// SIMATIC S7-200 project (STEP 7-Micro/WIN), CPU 226 REL 01.00

ORGANIZATION_BLOCK MAIN:OB1
TITLE= 项目注释：
// 
// 系统通过启动按钮1启动循环泵控制柜，控制循环泵1和循环泵2的运行，但循环泵1启动时，循环泵2不得同时运行，以避免电力过载。启动按钮3启动引风机控制柜，控制引风机；引风机启动前需确认循环泵运行标志置位，以确保炉内气流稳定。随后，鼓风机由启动按钮1触发，只有在引风机运行后才会启动，以维持炉内压力平衡。启动按钮2启动PLC控制柜，负责炉排电机、上煤电机、出渣电机和注油泵的运行。炉排电机由启动按钮2触发，需循环泵运行标志置位，以确保燃料供应；上煤电机只有在炉排电机运行后才会启动，以协调上煤和燃烧过程；出渣电机由启动按钮2控制，启动时不依赖炉排电机的状态。当上煤电机运行时，出渣电机可配合清除炉渣。注油泵在油压低时自动启动；延时定时器到时后，通过标志停止注油泵，以维持油压稳定。
// 系统通过多个传感器分别检测炉膛压力、炉膛温度、混合空气温度、排烟温度、进油温度和出油温度。当炉膛压力超过设定值时，触发报警标志；当炉膛温度高于设定值或低于设定值时，触发报警标志；炉膛温度低报警触发时，表示燃烧不足，上煤电机继续运行需谨慎。此时报警指示灯点亮；报警触发多个延时定时器，各定时器分别停止鼓风机、引风机、上煤电机和炉排电机，以安全停机。PID控制读取压力传感器和温度传感器的值，通过子程序调节炉膛压力和出油温度，确保工艺参数保持在设定范围内。操作员通过停止按钮1停止循环泵1，通过停止按钮2停止循环泵2；停止按钮3触发报警标志并点亮指示灯，保障操作安全。
// 
//  
BEGIN
Network 1 // 注油泵延时自动停止时间初始化
//  
// 
LD     SM0.1
MOVW   +1200, VW500
?000
Network 2 // 报警时间初始化
//  
// 
LD     SM0.1
MOVW   +300, VW502
Network 4 // 报警延时关断顺序初始化
// 
// 
LD     SM0.1
MOVW   +10, VW600
MOVW   +100, VW602
MOVW   +200, VW604
MOVW   +300, VW606
Network 5 // 报警延时关断顺序初始化
// 
// 
LDN    SM0.0
MOVW   +0, VW610
MOVW   +100, VW612
Network 7 // 炉膛报警压力设定
// 
// 
// 
LD     SM0.1
MOVW   -10000, VW1022
Network 8 // 炉膛报警温度高设定
// 
// 
LD     SM0.1
MOVW   +3000, VW1122
Network 9 // 炉膛报警温度低设定
// 
// 
// 
LD     SM0.1
MOVW   +1000, VW1124
Network 10 // 混合空气报警温度设定
// 
// 
LD     SM0.1
MOVW   +3000, VW1222
Network 11 // 排烟报警温度设定
// 
// 
LD     SM0.1
MOVW   +3000, VW1322
Network 12 // 出油报警温度高设定
// 
// 
// 
LD     SM0.1
MOVW   +3000, VW1522
Network 13 // 出油报警温度低设定
// 
// 
// 
LD     SM0.1
MOVW   +1000, VW1526
Network 15 // 模拟量设定值初始化--炉膛压力
// 
// 
LD     SM0.1
MOVW   -10000, VW1024
Network 16 // 模拟量设定值初始化--出油温度
// 
// 
LD     SM0.1
MOVW   +3000, VW1528
Network 18 // 循环泵控制柜－循环泵1
// 
// 
LD     I0.0
LPS
LD     M0.0
O      I0.3
O      T37
ALD
A      M0.2
AN     I0.5
AN     Q0.1
=      Q0.0
LPP
LPS
A      M0.0
S      M0.2, 1
LPP
A      M0.1
R      M0.2, 1
Network 19 // 泵1-延时等待运行信号
// 
// 
LD     Q0.0
EU
TOF    T37, +100
Network 20 // 循环泵控制柜－循环泵2
// 
// 
LD     I0.0
LPS
LD     M1.0
O      I0.4
O      T38
ALD
A      M1.2
AN     I0.6
AN     Q0.0
=      Q0.1
LPP
LPS
A      M1.0
S      M1.2, 1
LPP
A      M1.1
R      M1.2, 1
Network 21 // 泵2-延时等待运行信号
// 
// 
LD     Q0.1
EU
TOF    T38, +100
Network 22 // 循环泵启动信号
// 
// 
LD     Q0.0
O      Q0.1
=      M1.7
Network 24 // 引风机控制柜－引风机
// 
// 
LD     I0.2
LPS
LD     M2.0
O      I1.1
LDN    M2.1
O      Q0.5
ALD
ALD
AN     I1.2
A      M1.7
AN     T51
=      Q0.3
LPP
A      M2.2
=      Q0.2
Network 25 // 循环泵控制柜－鼓风机
//  
// 
//  
// 
LD     I0.0
LPS
LD     M3.0
O      I0.7
ALD
AN     M3.1
AN     I1.0
A      Q0.3
A      M1.7
AN     T50
=      Q0.5
LPP
A      M3.2
=      Q0.4
Network 27 // PLC控制柜－炉排电机
// 
// 
LD     I0.1
LD     M4.0
O      I2.0
ALD
LDN    M4.1
O      Q0.7
ALD
AN     I2.1
A      M1.7
AN     T53
=      Q0.6
Network 28 // PLC控制柜-上煤电机
// 
// 
LD     I0.1
LD     M5.0
O      I2.3
ALD
AN     M5.1
AN     I2.4
A      Q0.6
A      M1.7
AN     T52
=      Q0.7
Network 30 // PLC控制柜－出渣电机
// 
// 
LD     I0.1
LD     M6.0
O      I2.5
ALD
AN     M6.1
AN     I2.6
=      Q1.0
Network 31 // PLC控制柜－注油泵
// 
// 
LD     I0.1
LD     M7.0
O      I3.2
O      I3.1
ALD
AN     M7.1
AN     I3.3
AN     I3.0
AN     M7.7
=      Q1.1
Network 32
LD     I3.1
TOF    T39, VW500
Network 33
LD     T39
ED
=      M7.7
Network 35 // 模拟量读取/显示--炉膛压力
// 
// 
LDW<=  AIW4, +6500
MOVW   +6500, VW1000
Network 36
LDW>=  AIW4, +6500
AW<=   AIW4, +32000
MOVW   AIW4, VW1000
Network 37
LDW>=  AIW4, +32000
MOVW   +32000, VW1000
Network 38 // 炉膛压力线性运算
// 
// 
LD     SM0.0
MOVW   VW1000, VW1002
AENO
-I     +6500, VW1002
AENO
ITD    VW1002, VD1004
AENO
DTR    VD1004, VD1008
AENO
MOVR   VD1008, VD1012
AENO
/R     160.0, VD1012
AENO
ROUND  VD1012, VD1016
AENO
DTI    VD1016, VW1020
AENO
*I     -1, VW1020
Network 40 // 模拟量读取/显示--炉膛温度
// 
// 
LDW<=  AIW6, +6500
MOVW   +6500, VW1100
Network 41
LDW>=  AIW6, +6500
AW<=   AIW6, +32000
MOVW   AIW6, VW1100
Network 42
LDW>=  AIW6, +32000
MOVW   +32000, VW1100
Network 43 // 炉膛温度线性运算
// 
// 
// 
LD     SM0.0
MOVW   VW1100, VW1102
AENO
-I     +6500, VW1102
AENO
ITD    VW1102, VD1104
AENO
DTR    VD1104, VD1108
AENO
MOVR   VD1108, VD1112
AENO
/R     51.0, VD1112
AENO
ROUND  VD1112, VD1116
AENO
DTI    VD1116, VW1120
Network 45 // 模拟量读取/显示--混合空气温度
// 
// 
LDW<=  AIW8, +6500
MOVW   +6500, VW1200
Network 46
LDW>=  AIW8, +6500
AW<=   AIW8, +32000
MOVW   AIW8, VW1200
Network 47
LDW>=  AIW8, +32000
MOVW   +32000, VW1200
Network 48 // 炉膛温度线性运算
// 
// 
// 
LD     SM0.0
MOVW   VW1200, VW1202
AENO
-I     +6500, VW1202
AENO
ITD    VW1202, VD1204
AENO
DTR    VD1204, VD1208
AENO
MOVR   VD1208, VD1212
AENO
/R     51.0, VD1212
AENO
ROUND  VD1212, VD1216
AENO
DTI    VD1216, VW1220
Network 50 // 模拟量读取/显示--排烟温度
// 
// 
LDW<=  AIW10, +6500
MOVW   +6500, VW1300
Network 51
LDW>=  AIW10, +6500
AW<=   AIW10, +32000
MOVW   AIW10, VW1300
Network 52
LDW>=  AIW10, +32000
MOVW   +32000, VW1300
Network 53 // 排烟温度线性运算
// 
// 
// 
LD     SM0.0
MOVW   VW1300, VW1302
AENO
-I     +6500, VW1302
AENO
ITD    VW1302, VD1304
AENO
DTR    VD1304, VD1308
AENO
MOVR   VD1308, VD1312
AENO
/R     51.0, VD1312
AENO
ROUND  VD1312, VD1316
AENO
DTI    VD1316, VW1320
Network 55 // 模拟量读取/显示--进油温度
// 
// 
LDW<=  AIW12, +6500
MOVW   +6500, VW1400
Network 56
LDW>=  AIW12, +6500
AW<=   AIW12, +32000
MOVW   AIW12, VW1400
Network 57
LDW>=  AIW12, +32000
MOVW   +32000, VW1400
Network 58 // 进油温度线性运算
// 
// 
// 
LD     SM0.0
MOVW   VW1400, VW1402
AENO
-I     +6500, VW1402
AENO
ITD    VW1402, VD1404
AENO
DTR    VD1404, VD1408
AENO
MOVR   VD1408, VD1412
AENO
/R     51.0, VD1412
AENO
ROUND  VD1412, VD1416
AENO
DTI    VD1416, VW1420
Network 60 // 模拟量读取/显示--出油温度
// 
// 
LDW<=  AIW14, +6500
MOVW   +6500, VW1500
Network 61
LDW>=  AIW14, +6500
AW<=   AIW14, +32000
MOVW   AIW14, VW1500
Network 62
LDW>=  AIW14, +32000
MOVW   +32000, VW1500
Network 63 // 出油温度线性运算
// 
// 
// 
LD     SM0.0
MOVW   VW1500, VW1502
AENO
-I     +6500, VW1502
AENO
ITD    VW1502, VD1504
AENO
DTR    VD1504, VD1508
AENO
MOVR   VD1508, VD1512
AENO
/R     51.0, VD1512
AENO
ROUND  VD1512, VD1516
AENO
DTI    VD1516, VW1520
Network 65 // 炉膛负压报警控制
// 
// 
LDW>=  VW1020, VW1022
=      M8.0
Network 66
LDW<=  VW1022, -20000
=      M10.0
MOVW   -20000, VW1022
Network 67
LDW>=  VW1022, +0
=      M10.1
MOVW   +0, VW1022
Network 68 // 炉膛温度高报警控制
// 
// 
LDW>=  VW1120, VW1122
=      M8.1
Network 69
LDW>=  VW1122, +5000
=      M10.2
MOVW   +5000, VW1122
Network 70 // 炉膛温度低报警控制
// 
// 
LDW<=  VW1120, VW1124
=      M8.2
Network 71
LDW>=  VW1124, +5000
=      M10.3
MOVW   +5000, VW1224
Network 72
LDW>=  VW1124, VW1122
=      M10.4
MOVW   VW1122, VW1124
Network 73 // 混合空气温度报警控制
// 
// 
LDW>=  VW1220, VW1222
=      M8.3
Network 74
LDW>=  VW1222, +5000
=      M10.5
MOVW   +5000, VW1222
Network 75 // 排烟报警温度控制
// 
// 
LDW>=  VW1320, VW1322
=      M8.4
Network 76
LDW>=  VW1322, +5000
=      M10.6
MOVW   +5000, VW1322
Network 77 // 出油温度报警控制
// 
// 
LD     SM0.0
MOVW   VW1522, VW1524
+I     +6, VW1524
Network 78
// 
// 
LDW>=  VW1520, VW1524
=      M8.5
Network 79
LDW>=  VW1522, +5000
=      M10.7
MOVW   +5000, VW1522
Network 80
// 
// 
LDW<=  VW1520, VW1526
=      M8.6
Network 81
LDW>=  VW1526, +5000
=      M11.0
MOVW   +5000, VW1526
Network 82
LDW>=  VW1526, VW1522
=      M11.1
MOVW   VW1522, VW1526
Network 84 // 报警控制
// 
// 
LD     I0.5
EU
LD     I0.6
EU
OLD
LD     I1.0
EU
OLD
LD     I1.2
EU
OLD
LD     I1.5
EU
OLD
LD     I1.6
EU
OLD
LD     I2.1
EU
OLD
LD     I2.4
EU
OLD
LD     I2.6
EU
OLD
LD     I3.0
EU
OLD
LD     I3.1
EU
OLD
LD     I3.3
EU
OLD
LD     M8.0
EU
OLD
LD     M8.1
EU
OLD
LD     M8.2
EU
OLD
LD     M8.3
EU
OLD
LD     M8.4
EU
OLD
LD     M8.5
EU
OLD
LD     M8.6
EU
OLD
TOF    T40, VW502
S      M9.0, 1
Network 85 // 报警声音控制
// 
// 
LDN    T42
TON    T41, +10
Network 86
LD     T41
TON    T42, +10
Network 87 // 报警控制
// 
// 
LD     I0.5
O      I0.6
O      I1.0
O      I1.2
O      I1.5
O      I1.6
O      I2.1
O      I2.4
O      I2.6
O      I3.0
O      I3.1
O      I3.3
O      M8.0
O      M8.1
O      M8.2
O      M8.3
O      M8.4
O      M8.5
O      M8.6
A      M9.0
A      T40
AN     T42
=      Q1.2
Network 88 // 消音
// 
// 
LD     M9.1
R      M9.0, 1
Network 90 // 故障停机顺序
// 
// 
LD     M8.0
O      M8.1
O      M8.5
O      I1.5
O      I1.6
TON    T50, VW600
TON    T51, VW602
TON    T52, VW604
TON    T53, VW606
Network 91 // 进/出口油压高故障停机顺序控制
// 
// 
LDN    SM0.0
LD     I1.5
O      I1.6
ALD
TON    T55, VW610
TON    T56, VW612
Network 93 // PID模拟量设定值--炉膛压力设定
// 
// 
LD     SM0.0
ITD    VW1024, VD1026
AENO
DTR    VD1026, VD1030
AENO
MOVW   VW1030, VW104
/I     -20000, VW104
Network 94
LDW<=  VW1024, -20000
=      M11.2
MOVW   -20000, VW1024
Network 95
LDW>=  VW1024, +0
=      M11.3
MOVW   +0, VW1024
Network 96 // PID模拟量设定值--出油温度设定
// 
// 
LD     SM0.0
ITD    VW1528, VD1530
AENO
DTR    VD1530, VD1534
AENO
MOVW   VW1534, VW204
/I     +5000, VW204
Network 97
LDW>=  VW1528, +5000
=      M11.4
MOVW   +5000, VW1528
Network 99 // PID Kt 的几套参数 压力
// 
// 
LDW<   VW1020, -10000
MOVR   0.5, VD112
Network 100
LDW<=  VW1020, -10000
AW>=   VW1020, -20000
MOVR   0.3, VD112
Network 101
LDW>   VW1020, -20000
MOVR   0.2, VD112
Network 102 // PID Kt 的几套参数 炉膛温度高
// 
// 
LDW<   VW1520, +3000
MOVR   0.5, VD112
Network 103
LDW<=  VW1520, +3000
AW>=   VW1520, +4000
MOVR   0.3, VD112
Network 104
LDW>   VW1520, +4000
MOVR   0.2, VD112
Network 105 // PID调用
//  
// 
//  
// 
LD     SM0.1
CALL   SBR_0:SBR0
END_ORGANIZATION_BLOCK

SUBROUTINE_BLOCK SBR_0:SBR0
TITLE= 
// SUBROUTINE COMMENTS
// Press F1 for help and example program
//  
BEGIN
Network 1 // PID parameter 1
// VD100   过程变量PVn    0--1
// VD104   设定值SPn      0--1
// VD108   输出值Mn       0--1 （输入/输出）
// VD112   回路增益Kc
// VD116   采样时间Ts   second
// VD120   积分时间Ti   minute
// VD124   微分时间Td   minute
// VD128   积分项前项MX  0--1   （输入/输出）
// VD132   过程变量前值PVn-1  0--1   （输入/输出）
// 
LD     SM0.0
MOVR   0.0, VD100
MOVR   VD104, VD104
MOVR   0.0, VD108
MOVR   0.25, VD112
MOVR   0.1, VD116
MOVR   10.0, VD120
MOVR   0.0, VD124
Network 2 // PID parameter 2
// VD200   过程变量PVn    0--1
// VD204   设定值SPn      0--1
// VD208   输出值Mn       0--1 （输入/输出）
// VD212   回路增益Kc
// VD216   采样时间Ts   second
// VD220   积分时间Ti   minute
// VD224   微分时间Td   minute
// VD228   积分项前项MX  0--1   （输入/输出）
// VD232   过程变量前值PVn-1  0--1   （输入/输出）
// 
LD     SM0.0
MOVR   0.0, VD200
MOVR   VD204, VD204
MOVR   0.0, VD208
MOVR   0.25, VD212
MOVR   0.1, VD216
MOVR   10.0, VD220
MOVR   0.0, VD224
Network 3 // interrupt setting
// SMB34  interrupt 0 interval time=100 ms
// 
//  
// 
LD     SM0.0
MOVB   100, SMB34
AENO
ATCH   INT_0:INT0, 10
AENO
ENI
Network 28 // NETWORK TITLE (single line)
//  
// NETWORK COMMENTS
//  
// 
END_SUBROUTINE_BLOCK

INTERRUPT_BLOCK INT_0:INT0
TITLE= 
// INTERRUPT ROUTINE COMMENTS
// Press F1 for help and example program
//  
BEGIN
Network 1 // PV 转换成实数 1
// 把PV 存入累加器 AC0
// 32位整数转换成实数 存入 AC0 
// 标准化累加器中的值 存入 AC0
// 把标准化的PV值 存入 Table表
//  
// 
LD     SM0.0
ITD    AIW4, AC0
DTR    AC0, AC0
/R     32000.0, AC0
MOVR   AC0, VD100
Network 2 // PID AutoRun
// 当I0.1导通时 PID运行
// 
LD     I0.1
PID    VB100, 0
Network 3 // PID Out 1
// 
// 
LD     SM0.0
MOVR   VD108, AC0
*R     32000.0, AC0
ROUND  AC0, AC0
DTI    AC0, AC0
MOVW   AC0, AQW0
Network 4 // PV 转换成实数 2
// 把PV 存入累加器 AC0
// 32位整数转换成实数 存入 AC0 
// 标准化累加器中的值 存入 AC0
// 把标准化的PV值 存入 Table表
//  
// 
LD     SM0.0
ITD    AIW14, AC1
DTR    AC1, AC1
/R     32000.0, AC1
MOVR   AC1, VD200
Network 5 // PID AutoRun
// 当I0.1导通时 PID运行
// 
LD     I0.1
PID    VB200, 1
Network 6 // PID Out 2
// 
// 
LD     SM0.0
MOVR   VD208, AC1
*R     32000.0, AC1
ROUND  AC1, AC1
DTI    AC1, AC1
MOVW   AC1, AQW2
Network 29 // NETWORK TITLE (single line)
//  
// NETWORK COMMENTS
//  
// 
Network 54 // NETWORK TITLE (single line)
//  
// NETWORK COMMENTS
//  
// 
END_INTERRUPT_BLOCK
